FUNCTION FC_AnalogInputValueHandling
VAR_INPUT
	RowValue	:	WORD;	//Rohwert Sensor
	UpperLimit	:	REAL;	//Obere Grenze Umrechnungsbereich
	LowerLimit	:	REAL;	//Untere Grenze Umrechnungsbereich
END_VAR
VAR_OUTPUT
	ConvertedValue	:	REAL;	//Berechneter Wert
END_VAR
VAR
	tempConvertedRowValue	:	REAL;
	tempInputValueRange	:	REAL;
	tempCalculatedValue	:	REAL;
END_VAR

tempConvertedRowValue := TO_REAL(RowValue);
tempInputValueRange := tempConvertedRowValue / 100.0;
tempCalculatedValue := (tempInputValueRange * (UpperLimit - LowerLimit) / 10) + LowerLimit;

ConvertedValue := tempCalculatedValue;

END_FUNCTION

(* stored: Version 1.1.0.1
   POU FC_AnalogInputValueHandling: Id {7a3e07f7-bd82-4be6-b731-6cd987c87b4d}, SpecialFunc None *)
